PROGRAM Mobility
VAR
END_VAR

END_PROGRAM

(* stored: Version 1.1.0.1, ProductVersion 3.1.4022.18
   POU Mobility: Id {5e8d00ab-95b7-46ad-946e-67583346b988}, SpecialFunc None *)
